FUNCTION_BLOCK FB_TimerManager
VAR
	_aTimers: ARRAY [1..TIMERS.MAX_TIMER] OF I_Timer;
	_count: INT;
END_VAR

FOR

METHOD PUBLIC Register : BOOL
VAR_INPUT
	Timer: I_Timer;
END_VAR
END_METHOD

END_FUNCTION_BLOCK

(* stored: Version 1.1.0.1, ProductVersion 3.1.4024.10
   POU FB_TimerManager: Id {15ecb0f5-db53-447e-bb3c-cfce3e6e2076}, SpecialFunc None
   Method Register: Id {b01fc9cd-b3fe-43aa-adad-67ca8d1daf7f} *)
